Fanuc KAREL source: kt00261.KL

-- PROVISIONAL review KL for V1013-1; original PC SHA256 e704e86bb94d1db3bb9c3ae3290aae6c9949ffbd9700ed23dec27535eaf50221
-- Incomplete behavior may be omitted. Consult companion uncertainty JSON. Do not deploy.
PROGRAM KT00261
%NOLOCKGROUP
VAR
  R1 : REAL
  I2 : INTEGER
  OUT : BOOLEAN
BEGIN
  -- UNRESOLVED_PC offsets 5-16; opcodes 2E,23
  -- UNRESOLVED_PC offsets 21-32; opcodes 2E,23
  -- UNRESOLVED_PC offsets 37-57; opcodes 21,21,64,6D,23
  -- UNRESOLVED_PC offsets 62-66; opcodes 7F
END KT00261
